FUNCTION_BLOCK L1_Actuator
VAR CONSTANT
	COLOR_AAct 		: DWORD := 16#0000FF00;
	//COLOR_AIna 		: DWORD := 16#000000FF;
END_VAR

VAR_OUTPUT
	uiValue			: BOOL;					// Vinculación a la visualización
//	Name			: STRING; 				// Nombre del actuador, p.ej. K_1
	uiToolTip		: STRING;				// Tooltip en la visualización
END_VAR
VAR
	hwValue AT %Q*	: BOOL;					// Vinculación al hardware de la estación
	//dr				: REFERENCE TO L1_Director;
	
	//ETActive		: TIME;					// Valor de Clock.ET en el momento de la última activación
	//FPReloj			: R_TRIG;				// 
	//prValue			: BOOL := FALSE;		// Valor previo para detectar cambios de estado	
	//HasFailed		: BOOL := FALSE;		// El actuador ha fallado porque no ha terminado en tiempo
	(*
	uiEnabled		: BOOL := FALSE; 		// Deshabilitar el control cuando no está en modo manual
	uiColor			: DWORD := COLOR_AAct;	// Color por defecto rojo pálido
	uiInvisible		: BOOL := TRUE;			// Actuador gráfico invisible si no está pulsado
	uiUp			: REAL := 0;
	UIDown			: REAL := 0;
	uiLeft			: REAL := 0;
	uiRight			: REAL := 0;
	uiClockwise		: REAL := 0;
	uiUnclockwise	: REAL := 0; 
*)
	
END_VAR

METHOD ForceValue : BOOL
VAR_INPUT
	NewValue : BOOL;
END_VAR
uiValue := NewValue;
hwValue := NewValue;
END_METHOD

METHOD ProcessCycle : BOOL
VAR_INPUT
	gmMode		: L1_GEMMA;
	sfcValue 	: BOOL;		// estado del actuador devuelto por el Grafcet
END_VAR
IF gmMode = L1_GEMMA.F4VerificacionSinOrden THEN	
	hwValue := uiValue;	// Actualizar el hardware con la entrada desde la visualización
ELSE	
	hwValue := sfcValue; // Actualizar el hardware y la visualicación con la entrada desde el Grafcet
	uiValue := sfcValue;
END_IF
END_METHOD

END_FUNCTION_BLOCK

(* stored: Version 1.1.0.1, ProductVersion 3.1.4024.11
   POU L1_Actuator: Id {ad7a615f-d37f-4c2d-8af3-51dcf617a49f}, SpecialFunc None
   Method ForceValue: Id {289f89d6-23cc-4097-8d90-f6ae49e4f7e1}
   Method ProcessCycle: Id {ecf71777-ee3c-4e39-a4e9-a6f0d14f2603} *)
